//==================================================================================================
//							Beckhoff Automation Poland
//									30.03.2017
//		Mierzy czas zalaczenia wejscia. Podaje aktualny czas oraz czas ostatniego zalaczenia
//		W porownaniu do FB_TimeMeasure ma wejscie bReset
// 	v1.0 	|| TC v 3.1.4020.32		|| - pierwsza wersja
//==================================================================================================
FUNCTION_BLOCK FB_TimeMeasureEx
VAR_INPUT
	bOn										: BOOL;					// Zliczany sygnal
	bReset									: BOOL;					// Zerowanie wartosci
END_VAR
VAR_OUTPUT
	tCurrentTime							: TIME;
	tLastTime								: TIME;
END_VAR
VAR
	ton1									: TON;
	bOnOld									: BOOL;
END_VAR

IF bOn = FALSE AND bOnOld = TRUE THEN 
	tLastTime := tCurrentTime; 
END_IF
ton1(IN:= bOn, PT:= T#71582m47s295ms, Q=> , ET=> tCurrentTime);
bOnOld 						:= bOn;
IF bReset THEN
	bOnOld					:= FALSE;
	tLastTime				:= T#0S;
	tCurrentTime			:= T#0S;
	ton1(IN:= FALSE);
END_IF

END_FUNCTION_BLOCK

(* stored: Version 1.1.0.1, ProductVersion 3.1.4026.13, FileIdentifier f9c44413eabf5e5d46506d520b345bb2de4f7b48, FileSignature 319eb0a18f055ad8dc381aac2f5934a9428f2f7e22275bf69ba4e7069fd6f2887c465cec064fe9ebe5f923706c5290c3ae6e8764f85c936fe9bbc8d806136139b454240369806e4b77bbe82696aeaf15752c726e6be37dd949e93db31c3c7dd8492de29c0e11032ca8dfecb4a0f567b917982e9b09c587fbcaece4271e1ba81d7ef25dbaa1e3fe5949a03ed5dc9c573fb95b7524f4d404d1fd0eb1bb6b22fceafd0fb0a232c33e039bdc3458a5ee12fe47685210d5c8f25de9e6c209c0e6c6567364c097aa976f63515a3a4e9ca1492e71dcd28a85869f2cb7013cf827d870a1b86785c8b2bacc3c167f83a822421c6326deb0b69ddbbd19b29e94bc91ac20c0
   POU FB_TimeMeasureEx: Id {577c1614-5184-4c84-bd6f-a25228b68a60}, SpecialFunc None *)
